SUBAPPLICATION AX_MIN_TP (* Minimum-Pulsbreite: AX_Q folgt AX_IN, ist aber mindestens PT lang - kuerzere Pulse werden auf PT gestreckt, laengere Pulse unveraendert durchgereicht (Gegenstueck zu AX_TP, das immer exakt PT macht, und AX_TLIM, das auf maximal PT kappt). Franz: Bunkerboden-Vorlauf im Automatikbetrieb braucht eine Mindestzeit. Sicherheitshinweis (Martin Schuder): dieser Baustein selbst hat KEINEN Hard-Abbruch - ein Endschalter, der den Puls jederzeit sofort unterbrechen soll, muss extern per AX_AND(AX_Q, NOT Endschalter) NACH diesem Baustein verknuepft werden, nicht ueber diesen Baustein selbst. *)
  (* Standard: 61499-2; Description: Copyright (c) 2026 Meisterschulen am Ostbahnhof This program and the accompanying materials are made available under the terms of the Eclipse Public License 2.0 which is available at https://www.eclipse.org/legal/epl-2.0/ SPDX-License-Identifier: EPL-2.0 *)
  (* Version 1.2, 2026-09-29, Franz Höpfinger, Meisterschulen am Ostbahnhof, Franz-Vereinfachung (verworfen: v1.1 mit ACTIVE/AX_TON/AX_R_TRIG-Latch-Konstruktion): AX_Q = AX_IN OR AX_TP_MinZeit.Q reicht - AX_TP ist non-retriggerable und laeuft nach der steigenden Flanke von AX_IN immer exakt PT durch, egal ob AX_IN vorher schon wieder abfaellt. Kuerzere Pulse werden dadurch automatisch auf PT gestreckt (AX_TP.Q haelt bis PT), laengere Pulse bleiben unveraendert (AX_IN selbst haelt Q hoch, auch nachdem AX_TP.Q laengst auf PT abgelaufen ist). Kein Latch, kein AX_TON noetig. Neuer SubAppEventInput R (Reset) auf AX_TP.R durchgereicht. *)
  (* Version 1.1, 2026-09-29, Franz Höpfinger, Meisterschulen am Ostbahnhof, Franz: 'sind in allen Faellen E_SWITCH richtig, oder waere es ein R_TRIG und F_TRIG?' - komplett neu, ohne E_SWITCH/E_RF_TRIG/rohe E_-Bausteine: durchgehend das im Projekt etablierte AX-Adapter-Idiom. Reset-Bedingung ist ein simples AX_AND (NOT(AX_IN) AND AX_TON.Q, wobei AX_TON an ACTIVE.Q haengt - 'seit mindestens PT aktiv'), dessen steigende Flanke (AX_R_TRIG) ACTIVE.R ausloest, egal welche der beiden Seiten zuletzt eintrifft. Bleibt komplett auf Adapter-Ebene, keine IN_TO_BOOL/BOOL_TO_Q-Konverter mehr noetig. (Verworfen, siehe v1.2 - noch einfacher.) *)
  (* Version 1.0, 2026-09-29, Franz Höpfinger, Meisterschulen am Ostbahnhof, initial implementation (verworfen, siehe v1.1) - E_SWITCH-basiert. *)
  PACKAGE adapter::events::unidirectional::timers;
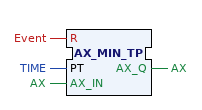
  EVENT_INPUT
    R; (* Reset *)
  END_EVENT
  VAR_INPUT
    PT : TIME; (* Mindest-Pulsbreite *)
  END_VAR
  SOCKETS
    AX_IN : adapter::types::unidirectional::AX; (* Roher Eingangspuls *)
  END_SOCKETS
  PLUGS
    AX_Q : adapter::types::unidirectional::AX; (* Auf mindestens PT gestreckter Ausgang *)
  END_PLUGS
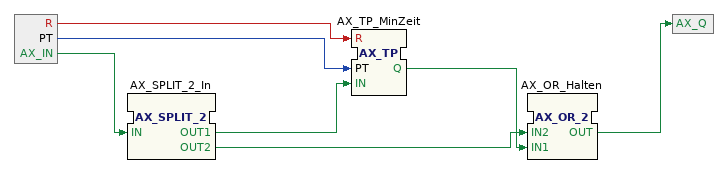
  FBS
    AX_SPLIT_2_In : adapter::events::unidirectional::AX_SPLIT_2; (* AX_IN wird fuer AX_TP_MinZeit.IN UND direkt fuer AX_OR_Halten gebraucht *)
    AX_TP_MinZeit : adapter::events::unidirectional::timers::AX_TP; (* Non-retriggerable - laeuft nach der steigenden Flanke von AX_IN immer exakt PT durch, unabhaengig davon ob AX_IN vorher schon wieder abfaellt *)
    AX_OR_Halten : adapter::booleanOperators::AX_OR_2; (* AX_IN OR AX_TP_MinZeit.Q - haelt den Ausgang, solange entweder der rohe Puls noch da ist (laengere Pulse) oder die Mindestzeit noch laeuft (kuerzere Pulse) *)
  END_FBS
  EVENT_CONNECTIONS
    R TO AX_TP_MinZeit.R;
  END_CONNECTIONS
  DATA_CONNECTIONS
    PT TO AX_TP_MinZeit.PT;
  END_CONNECTIONS
  ADAPTER_CONNECTIONS
    AX_IN TO AX_SPLIT_2_In.IN;
    AX_SPLIT_2_In.OUT1 TO AX_TP_MinZeit.IN;
    AX_SPLIT_2_In.OUT2 TO AX_OR_Halten.IN2;
    AX_TP_MinZeit.Q TO AX_OR_Halten.IN1;
    AX_OR_Halten.OUT TO AX_Q;
  END_CONNECTIONS
END_SUBAPPLICATION
